TYPE ST_LaudaCommands :
STRUCT
	Read	: ST_LaudaReadCommands;
	Write	: ST_LaudaWriteCommands;
END_STRUCT
END_TYPE

(* stored: Version 1.1.0.1, ProductVersion 3.1.4024.13
   DUT ST_LaudaCommands: Id {58f56184-a241-44f5-bdb2-48de90ce09c9} *)
